INTERFACE I_HomingStrategy EXTENDS I_MotionSequence

END_INTERFACE

(* stored: Version 1.1.0.1, ProductVersion 3.1.4024.15
   Itf I_HomingStrategy: Id {a5a9bf4a-8f58-4ca6-b0a2-b32da40ca435} *)
